FUNCTION F_PB_GetTransportControlDataRef : REFERENCE TO ST_TransportControlData
(**************************************************************************************
 * 	Application		:	BoxControl Framework
 *	Revision		:	$Revision:  $
 *	Revision date	:	$Date: $
 *	Last changed by	:	$Author: q8sheds $
 *	URL				:	$URL: $
 *
 *	Purpose			:	return Transport control data as reference
 *
 * ------------------------------------------------------------------------------------
 *	Copyright Swisslog [IP AG], Switzerland. All rights reserved.
 * 
 * ------------------------------------------------------------------------------------
 *	
 * 	Revision History: 
 *
 * 	VERSION			DATE			INITIALS			DESCRIPTION
 *	0.1				01.01.2001		swl					Example
 *
 **************************************************************************************)
VAR_INPUT
	eFunctionNumber		: E_FunctionNumber; // Function number
	ZoneNumber			: INT; // Zone number
END_VAR

//init
F_PB_GetTransportControlDataRef REF= PBTransportCtrl.pbTransportControlDataEmpty;	//return ref to empty transportcontroller data to avoid reutrn of NULL

// Check if function number is valid
IF(  eFunctionNumber > E_FunctionNumber.F_BEGIN_FUNCTION AND eFunctionNumber < E_FunctionNumber.F_END_FUNCTION AND
	 ZoneNumber > 0 AND ZoneNumber <= NUMBER_OF_ZONES_PER_FUNCTION) THEN
	// Check reference is valid
	IF __ISVALIDREF(FunctionRegistry[eFunctionNumber].Zone[ZoneNumber].refZoneData) THEN
   		// Return transport control data   				
		F_PB_GetTransportControlDataRef REF= FunctionRegistry[eFunctionNumber].Zone[ZoneNumber].refZoneData.TransportControlData;
	END_IF
END_IF

END_FUNCTION

(* stored: Version 1.1.0.1, ProductVersion 3.1.4022.12
   POU F_PB_GetTransportControlDataRef: Id {5740b59b-3ef0-4fe9-908b-47eb9cc809bd}, SpecialFunc None *)
